PROGRAM Q1_MOTOR
VAR
	ClearFault: FB_ClearFault;
	SetEnableState: FB_SetEnableState;
	SetHomingParameter: FB_SetHomingParameter;
	FindHome: FB_FindHome;
	SetMotorParameter: FB_SetMotorParameter;
	SetPositionProfile: FB_SetPositionProfile;
	SetOperationMode: FB_SetOperationMode;
	MoveToPosition: FB_MoveToPosition;
	GetMovementState: FB_GetMovementState;
	SetDisableState: FB_SetDisableState;
	SetPositionMust: FB_SetPositionMust;
	POSITION: DINT;
END_VAR

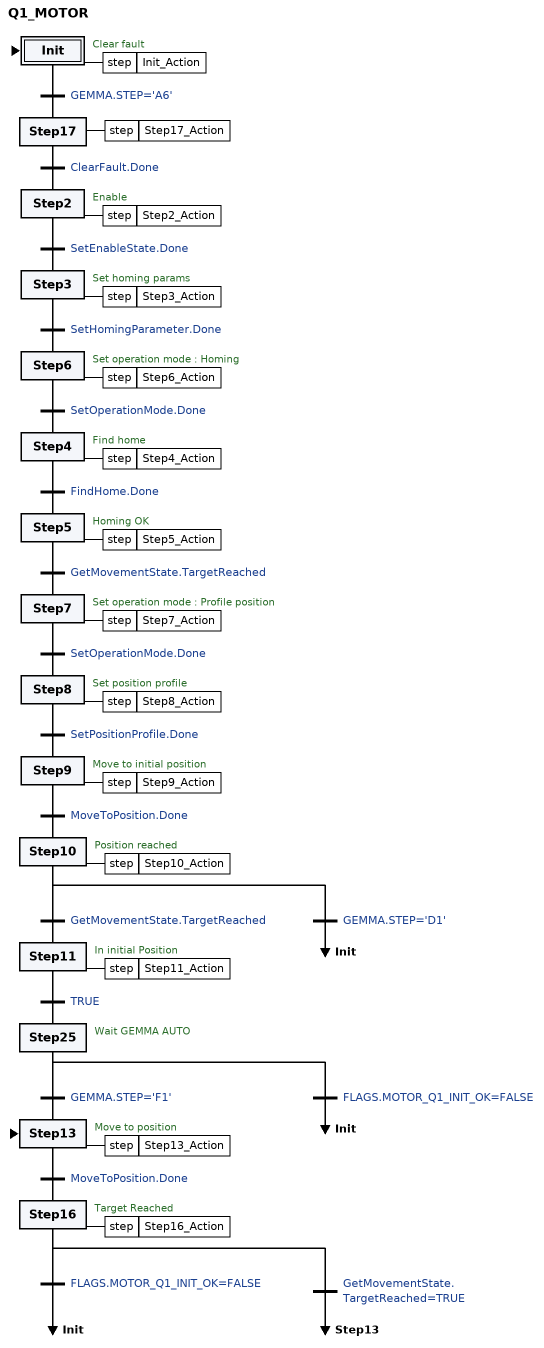
// Clear fault
INITIAL_STEP Init:
    Init_Action(N);  // step action
END_STEP
TRANSITION FROM Init TO Step17
    := GEMMA.STEP='A6';
END_TRANSITION
STEP Step17:
    Step17_Action(N);  // step action
END_STEP
TRANSITION FROM Step17 TO Step2
    := ClearFault.Done;
END_TRANSITION
// Enable
STEP Step2:
    Step2_Action(N);  // step action
END_STEP
TRANSITION FROM Step2 TO Step3
    := SetEnableState.Done;
END_TRANSITION
// Set homing params
STEP Step3:
    Step3_Action(N);  // step action
END_STEP
TRANSITION FROM Step3 TO Step6
    := SetHomingParameter.Done;
END_TRANSITION
// Set operation mode : Homing
STEP Step6:
    Step6_Action(N);  // step action
END_STEP
TRANSITION FROM Step6 TO Step4
    := SetOperationMode.Done;
END_TRANSITION
// Find home
STEP Step4:
    Step4_Action(N);  // step action
END_STEP
TRANSITION FROM Step4 TO Step5
    := FindHome.Done;
END_TRANSITION
// Homing OK
STEP Step5:
    Step5_Action(N);  // step action
END_STEP
TRANSITION FROM Step5 TO Step7
    := GetMovementState.TargetReached;
END_TRANSITION
// Set operation mode : Profile position
STEP Step7:
    Step7_Action(N);  // step action
END_STEP
TRANSITION FROM Step7 TO Step8
    := SetOperationMode.Done;
END_TRANSITION
// Set position profile
STEP Step8:
    Step8_Action(N);  // step action
END_STEP
TRANSITION FROM Step8 TO Step9
    := SetPositionProfile.Done;
END_TRANSITION
// Move to initial position
STEP Step9:
    Step9_Action(N);  // step action
END_STEP
TRANSITION FROM Step9 TO Step10
    := MoveToPosition.Done;
END_TRANSITION
// Position reached
STEP Step10:
    Step10_Action(N);  // step action
END_STEP
TRANSITION FROM Step10 TO Step11
    := GetMovementState.TargetReached;
END_TRANSITION
TRANSITION FROM Step10 TO Init
    := GEMMA.STEP='D1';
END_TRANSITION
// In initial Position
STEP Step11:
    Step11_Action(N);  // step action
END_STEP
TRANSITION FROM Step11 TO Step25
    := TRUE;
END_TRANSITION
// Wait GEMMA AUTO
STEP Step25:
END_STEP
TRANSITION FROM Step25 TO Step13
    := GEMMA.STEP='F1';
END_TRANSITION
TRANSITION FROM Step25 TO Init
    := FLAGS.MOTOR_Q1_INIT_OK=FALSE;
END_TRANSITION
// Move to position
STEP Step13:
    Step13_Action(N);  // step action
END_STEP
TRANSITION FROM Step13 TO Step16
    := MoveToPosition.Done;
END_TRANSITION
// Target Reached
STEP Step16:
    Step16_Action(N);  // step action
END_STEP
TRANSITION FROM Step16 TO Init
    := FLAGS.MOTOR_Q1_INIT_OK=FALSE;
END_TRANSITION
TRANSITION FROM Step16 TO Step13
    := GetMovementState.TargetReached=TRUE;
END_TRANSITION

ACTION Step10_Action:
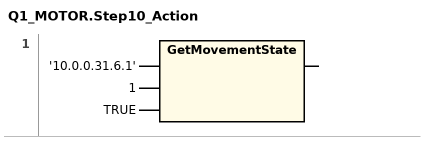
// NETWORK 1
GetMovementState('10.0.0.31.6.1', 1, TRUE);
END_ACTION

ACTION Step17_Action:
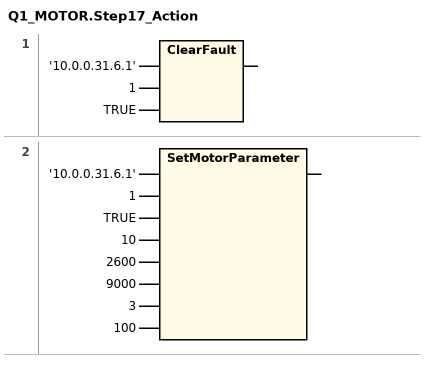
// NETWORK 1
ClearFault('10.0.0.31.6.1', 1, TRUE);

// NETWORK 2
SetMotorParameter('10.0.0.31.6.1', 1, TRUE, 10, 2600, 9000, 3, 100);
END_ACTION

ACTION Step13_Action:
(*Limitation deplacement Moteur*)
IF FLAGS.MOTOR_Q1_POSITION>MOTOR_Q1_POSITION_MAX THEN
	POSITION:=MOTOR_Q1_POSITION_MAX;
ELSIF FLAGS.MOTOR_Q1_POSITION<0 THEN
	POSITION:=0;
ELSE
	POSITION:=FLAGS.MOTOR_Q1_POSITION;
END_IF


MoveToPosition(
	ADSNetId:= '10.0.0.31.6.1',
	NodeId:= 1,
	Write:= TRUE,
	TargetPosition:= POSITION,
	Absolut:= TRUE);
END_ACTION

ACTION Step8_Action:
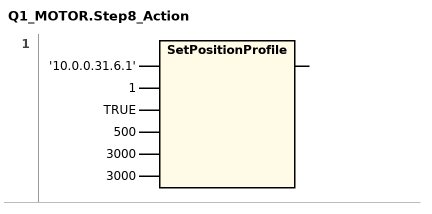
// NETWORK 1
SetPositionProfile('10.0.0.31.6.1', 1, TRUE, 500, 3000, 3000);
END_ACTION

ACTION Step16_Action:
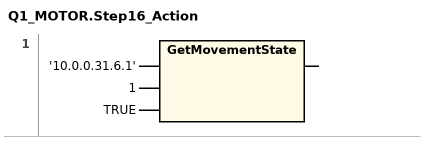
// NETWORK 1
GetMovementState('10.0.0.31.6.1', 1, TRUE);
END_ACTION

ACTION Step4_Action:
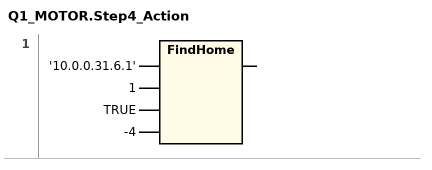
// NETWORK 1
FindHome('10.0.0.31.6.1', 1, TRUE, -4);
END_ACTION

ACTION Step3_Action:
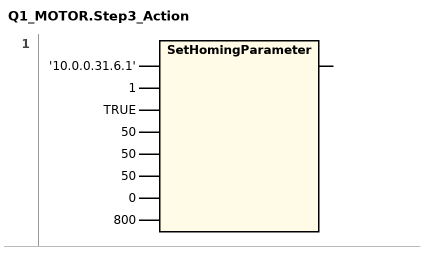
// NETWORK 1
SetHomingParameter('10.0.0.31.6.1', 1, TRUE, 50, 50, 50, 0, 800);
END_ACTION

ACTION Step5_Action:
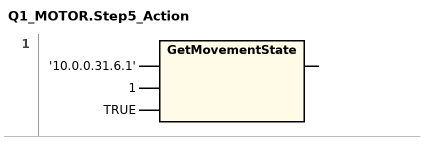
// NETWORK 1
GetMovementState('10.0.0.31.6.1', 1, TRUE);
END_ACTION

ACTION Step2_Action:
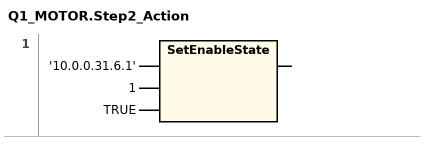
// NETWORK 1
SetEnableState('10.0.0.31.6.1', 1, TRUE);
END_ACTION

ACTION Init_Action:

END_ACTION

ACTION Step6_Action:
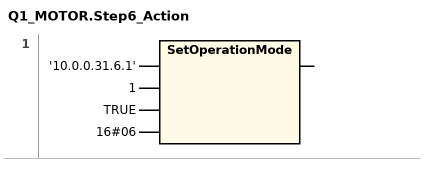
// NETWORK 1
SetOperationMode('10.0.0.31.6.1', 1, TRUE, 16#06);
END_ACTION

ACTION Step11_Action:

(*SetDisableState(
	ADSNetId:= '10.0.0.31.6.1',
	NodeId:= 1,
	Write:= TRUE);*)

FLAGS.MOTOR_Q1_INIT_OK:=TRUE;
END_ACTION

ACTION Step7_Action:
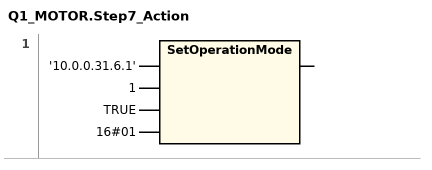
// NETWORK 1
SetOperationMode('10.0.0.31.6.1', 1, TRUE, 16#01);
END_ACTION

ACTION Step9_Action:
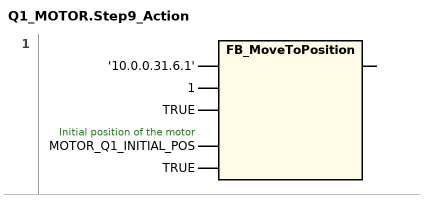
// NETWORK 1
//   MOTOR_Q1_INITIAL_POS: Initial position of the motor
FB_MoveToPosition('10.0.0.31.6.1', 1, TRUE, MOTOR_Q1_INITIAL_POS, TRUE);
END_ACTION

END_PROGRAM

(* stored: Version 1.1.0.1, ProductVersion 3.1.0.26
   POU Q1_MOTOR: Id {0f7f50a6-4eb5-48ae-becf-0f2f83018cab}
   Action Step10_Action: Id {194456a4-efae-460f-ac18-c896b13eff8f}
   Action Step17_Action: Id {23b68f97-cbc0-4c46-9b49-4b53341d0234}
   Action Step13_Action: Id {296f0c86-f375-4890-bef5-9c8d690ef396}
   Action Step8_Action: Id {3e513f0e-7bfb-48c9-a4ae-590b86852a52}
   Action Step16_Action: Id {4414d5c5-de3e-43d9-a6e2-c5ed6e6cbc79}
   Action Step4_Action: Id {4fdbe497-f540-42d9-b230-bc3f68374596}
   Action Step3_Action: Id {5f3735fb-0590-4cd0-a0ea-305db6bf34fd}
   Action Step5_Action: Id {61e0c32d-87c4-4da6-ac15-9157af4ca9e3}
   Action Step2_Action: Id {9ee61bc4-474a-47eb-ae49-b47f78eb9ad0}
   Action Init_Action: Id {a225051f-b32c-4844-8673-b4efebb19f2f}
   Action Step6_Action: Id {a7834f00-744c-4b35-9300-de5a17aa8f49}
   Action Step11_Action: Id {cdc65f18-e940-47cc-ac52-ae09e51b751a}
   Action Step7_Action: Id {dad494ec-eac8-47d4-87e3-ef9dea8b3b5d}
   Action Step9_Action: Id {ecc06163-9d5a-47b0-bab8-a5184ba20d50} *)
